PROGRAM FermentationProcess_001
VAR
	

	//MCC Driver	
	fbDriveReverse_001		      : FB_DriveReverse;
	fbDriveReverse_002		      : FB_DriveReverse;
	fbDriveReverse_003		      : FB_DriveReverse;
	fbDriveReverse_004		      : FB_DriveReverse;
	fbDriveReverse_005		      : FB_DriveReverse;
	fbDriveReverse_006		      : FB_DriveReverse;
	fbDriveReverse_007		      : FB_DriveReverse;
	fbDriveReverse_008		      : FB_DriveReverse;
	fbDriveReverse_009		      : FB_DriveReverse;
	fbDriveReverse_010		      : FB_DriveReverse;
	fbDriveReverse_011		      : FB_DriveReverse;
	fbDriveReverse_012		      : FB_DriveReverse;
	fbDriveReverse_013		      : FB_DriveReverse;
	fbDriveReverse_014		      : FB_DriveReverse;
	fbDriveReverse_015		      : FB_DriveReverse;
	fbDriveReverse_016		      : FB_DriveReverse;
	fbDriveReverse_017		      : FB_DriveReverse;
	fbDriveReverse_018		      : FB_DriveReverse;
	fbDriveReverse_019		      : FB_DriveReverse;
	fbDriveReverse_020		      : FB_DriveReverse;


	//MCC Driver Control
	fbMccRev_001			 	  : FB_MotorControlReverse(fbDriveReverse_001);
	fbMccRev_002			 	  : FB_MotorControlReverse(fbDriveReverse_002);
	fbMccRev_003			 	  : FB_MotorControlReverse(fbDriveReverse_003);
	fbMccRev_004 	 			  : FB_MotorControlReverse(fbDriveReverse_004);
	fbMccRev_005			 	  : FB_MotorControlReverse(fbDriveReverse_005);
	fbMccRev_006			 	  : FB_MotorControlReverse(fbDriveReverse_006);
	fbMccRev_007				  : FB_MotorControlReverse(fbDriveReverse_007);
	fbMccRev_008 	 			  : FB_MotorControlReverse(fbDriveReverse_008);
	fbMccRev_009 	  			  : FB_MotorControlReverse(fbDriveReverse_009);
	fbMccRev_010 	              : FB_MotorControlReverse(fbDriveReverse_010);
	fbMccRev_011			 	  : FB_MotorControlReverse(fbDriveReverse_011);
	fbMccRev_012			 	  : FB_MotorControlReverse(fbDriveReverse_012);
	fbMccRev_013			 	  : FB_MotorControlReverse(fbDriveReverse_013);
	fbMccRev_014 	 			  : FB_MotorControlReverse(fbDriveReverse_014);
	fbMccRev_015			 	  : FB_MotorControlReverse(fbDriveReverse_015);
	fbMccRev_016			 	  : FB_MotorControlReverse(fbDriveReverse_016);
	fbMccRev_017				  : FB_MotorControlReverse(fbDriveReverse_017);
	fbMccRev_018 	 			  : FB_MotorControlReverse(fbDriveReverse_018);
	fbMccRev_019 	  			  : FB_MotorControlReverse(fbDriveReverse_019);
	fbMccRev_020 	              : FB_MotorControlReverse(fbDriveReverse_020);
	
	//Temperature Sensor
	fbTempSens_001				  : FB_Scaling;
	fbTempSens_002				  : FB_Scaling;
	fbTempSens_003				  : FB_Scaling;
	//Level Sensor
	fbLevelSens_001				  : FB_Scaling;
	//Ph Sensor
	fbPhSens_001				  : FB_Scaling;	
	//Pressure Sensor
	fbPressureSens_001			  : FB_Scaling;	
	
	
	
	
	
END_VAR

ACT_Motor();
ACT_TempSens();
ACT_LevelSens();
ACT_PhSens();

ACTION ACT_LevelSens:
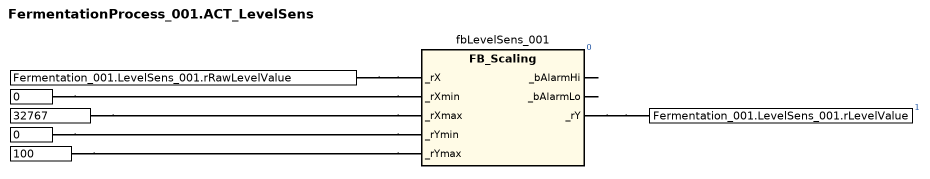
fbLevelSens_001(
    _rX := Fermentation_001.LevelSens_001.rRawLevelValue,
    _rXmin := 0,
    _rXmax := 32767,
    _rYmin := 0,
    _rYmax := 100); // FB_Scaling
Fermentation_001.LevelSens_001.rLevelValue := fbLevelSens_001._rY;
END_ACTION

ACTION ACT_Motor:
//Sygnały obiektów MccRev_* mieszadeł fermentora

//***************************************************SCADA********************************************************

//MccRev_001 variable sets by SCADA
FermentationProcess_001.fbMccRev_001.ScadaAutoButton     := Fermentation_001.MccRev_001.bAutoButton;    // SCADA button Auto Command
FermentationProcess_001.fbMccRev_001.ScadaForwardButton  := Fermentation_001.MccRev_001.bForwardButton; // SCADA button Forward Command
FermentationProcess_001.fbMccRev_001.ScadaReverseButton  := Fermentation_001.MccRev_001.bReverseButton; // SCADA button Reverse Command

//MccRev_002 variable sets by SCADA
FermentationProcess_001.fbMccRev_002.ScadaAutoButton     := Fermentation_001.MccRev_002.bAutoButton;    // SCADA button Auto Command
FermentationProcess_001.fbMccRev_002.ScadaForwardButton  := Fermentation_001.MccRev_002.bForwardButton; // SCADA button Forward Command
FermentationProcess_001.fbMccRev_002.ScadaReverseButton  := Fermentation_001.MccRev_002.bReverseButton; // SCADA button Reverse Command

//MccRev_003 variable sets by SCADA
FermentationProcess_001.fbMccRev_003.ScadaAutoButton     := Fermentation_001.MccRev_003.bAutoButton;    // SCADA button Auto Command
FermentationProcess_001.fbMccRev_003.ScadaForwardButton  := Fermentation_001.MccRev_003.bForwardButton; // SCADA button Forward Command
FermentationProcess_001.fbMccRev_003.ScadaReverseButton  := Fermentation_001.MccRev_003.bReverseButton; // SCADA button Reverse Command

//MccRev_004 variable sets by SCADA
FermentationProcess_001.fbMccRev_004.ScadaAutoButton     := Fermentation_001.MccRev_004.bAutoButton;    // SCADA button Auto Command
FermentationProcess_001.fbMccRev_004.ScadaForwardButton  := Fermentation_001.MccRev_004.bForwardButton; // SCADA button Forward Command
FermentationProcess_001.fbMccRev_004.ScadaReverseButton  := Fermentation_001.MccRev_004.bReverseButton; // SCADA button Reverse Command

//MccRev_005 variable sets by SCADA
FermentationProcess_001.fbMccRev_005.ScadaAutoButton     := Fermentation_001.MccRev_005.bAutoButton;    // SCADA button Auto Command
FermentationProcess_001.fbMccRev_005.ScadaForwardButton  := Fermentation_001.MccRev_005.bForwardButton; // SCADA button Forward Command
FermentationProcess_001.fbMccRev_005.ScadaReverseButton  := Fermentation_001.MccRev_005.bReverseButton; // SCADA button Reverse Command

//MccRev_006 variable sets by SCADA
FermentationProcess_001.fbMccRev_006.ScadaAutoButton     := Fermentation_001.MccRev_006.bAutoButton;    // SCADA button Auto Command
FermentationProcess_001.fbMccRev_006.ScadaForwardButton  := Fermentation_001.MccRev_006.bForwardButton; // SCADA button Forward Command
FermentationProcess_001.fbMccRev_006.ScadaReverseButton  := Fermentation_001.MccRev_006.bReverseButton; // SCADA button Reverse Command

//MccRev_007 variable sets by SCADA
FermentationProcess_001.fbMccRev_007.ScadaAutoButton     := Fermentation_001.MccRev_007.bAutoButton;    // SCADA button Auto Command
FermentationProcess_001.fbMccRev_007.ScadaForwardButton  := Fermentation_001.MccRev_007.bForwardButton; // SCADA button Forward Command
FermentationProcess_001.fbMccRev_007.ScadaReverseButton  := Fermentation_001.MccRev_007.bReverseButton; // SCADA button Reverse Command

//MccRev_008 variable sets by SCADA
FermentationProcess_001.fbMccRev_008.ScadaAutoButton     := Fermentation_001.MccRev_008.bAutoButton;    // SCADA button Auto Command
FermentationProcess_001.fbMccRev_008.ScadaForwardButton  := Fermentation_001.MccRev_008.bForwardButton; // SCADA button Forward Command
FermentationProcess_001.fbMccRev_008.ScadaReverseButton  := Fermentation_001.MccRev_008.bReverseButton; // SCADA button Reverse Command

//MccRev_009 variable sets by SCADA
FermentationProcess_001.fbMccRev_009.ScadaAutoButton     := Fermentation_001.MccRev_009.bAutoButton;    // SCADA button Auto Command
FermentationProcess_001.fbMccRev_009.ScadaForwardButton  := Fermentation_001.MccRev_009.bForwardButton; // SCADA button Forward Command
FermentationProcess_001.fbMccRev_009.ScadaReverseButton  := Fermentation_001.MccRev_009.bReverseButton; // SCADA button Reverse Command

//MccRev_010 variable sets by SCADA
FermentationProcess_001.fbMccRev_010.ScadaAutoButton     := Fermentation_001.MccRev_010.bAutoButton;    // SCADA button Auto Command
FermentationProcess_001.fbMccRev_010.ScadaForwardButton  := Fermentation_001.MccRev_010.bForwardButton; // SCADA button Forward Command
FermentationProcess_001.fbMccRev_010.ScadaReverseButton  := Fermentation_001.MccRev_010.bReverseButton; // SCADA button Reverse Command

//MccRev_011 variable sets by SCADA
FermentationProcess_001.fbMccRev_011.ScadaAutoButton     := Fermentation_001.MccRev_011.bAutoButton;    // SCADA button Auto Command
FermentationProcess_001.fbMccRev_011.ScadaForwardButton  := Fermentation_001.MccRev_011.bForwardButton; // SCADA button Forward Command
FermentationProcess_001.fbMccRev_011.ScadaReverseButton  := Fermentation_001.MccRev_011.bReverseButton; // SCADA button Reverse Command

//MccRev_012 variable sets by SCADA
FermentationProcess_001.fbMccRev_012.ScadaAutoButton     := Fermentation_001.MccRev_012.bAutoButton;    // SCADA button Auto Command
FermentationProcess_001.fbMccRev_012.ScadaForwardButton  := Fermentation_001.MccRev_012.bForwardButton; // SCADA button Forward Command
FermentationProcess_001.fbMccRev_012.ScadaReverseButton  := Fermentation_001.MccRev_012.bReverseButton; // SCADA button Reverse Command

//MccRev_013 variable sets by SCADA
FermentationProcess_001.fbMccRev_013.ScadaAutoButton     := Fermentation_001.MccRev_013.bAutoButton;    // SCADA button Auto Command
FermentationProcess_001.fbMccRev_013.ScadaForwardButton  := Fermentation_001.MccRev_013.bForwardButton; // SCADA button Forward Command
FermentationProcess_001.fbMccRev_013.ScadaReverseButton  := Fermentation_001.MccRev_013.bReverseButton; // SCADA button Reverse Command

//MccRev_014 variable sets by SCADA
FermentationProcess_001.fbMccRev_014.ScadaAutoButton     := Fermentation_001.MccRev_014.bAutoButton;    // SCADA button Auto Command
FermentationProcess_001.fbMccRev_014.ScadaForwardButton  := Fermentation_001.MccRev_014.bForwardButton; // SCADA button Forward Command
FermentationProcess_001.fbMccRev_014.ScadaReverseButton  := Fermentation_001.MccRev_014.bReverseButton; // SCADA button Reverse Command

//MccRev_015 variable sets by SCADA
FermentationProcess_001.fbMccRev_015.ScadaAutoButton     := Fermentation_001.MccRev_015.bAutoButton;    // SCADA button Auto Command
FermentationProcess_001.fbMccRev_015.ScadaForwardButton  := Fermentation_001.MccRev_015.bForwardButton; // SCADA button Forward Command
FermentationProcess_001.fbMccRev_015.ScadaReverseButton  := Fermentation_001.MccRev_015.bReverseButton; // SCADA button Reverse Command

//MccRev_016 variable sets by SCADA
FermentationProcess_001.fbMccRev_016.ScadaAutoButton     := Fermentation_001.MccRev_016.bAutoButton;    // SCADA button Auto Command
FermentationProcess_001.fbMccRev_016.ScadaForwardButton  := Fermentation_001.MccRev_016.bForwardButton; // SCADA button Forward Command
FermentationProcess_001.fbMccRev_016.ScadaReverseButton  := Fermentation_001.MccRev_016.bReverseButton; // SCADA button Reverse Command

//MccRev_017 variable sets by SCADA
FermentationProcess_001.fbMccRev_017.ScadaAutoButton     := Fermentation_001.MccRev_017.bAutoButton;    // SCADA button Auto Command
FermentationProcess_001.fbMccRev_017.ScadaForwardButton  := Fermentation_001.MccRev_017.bForwardButton; // SCADA button Forward Command
FermentationProcess_001.fbMccRev_017.ScadaReverseButton  := Fermentation_001.MccRev_017.bReverseButton; // SCADA button Reverse Command

//MccRev_018 variable sets by SCADA
FermentationProcess_001.fbMccRev_018.ScadaAutoButton     := Fermentation_001.MccRev_018.bAutoButton;    // SCADA button Auto Command
FermentationProcess_001.fbMccRev_018.ScadaForwardButton  := Fermentation_001.MccRev_018.bForwardButton; // SCADA button Forward Command
FermentationProcess_001.fbMccRev_018.ScadaReverseButton  := Fermentation_001.MccRev_018.bReverseButton; // SCADA button Reverse Command

//MccRev_019 variable sets by SCADA
FermentationProcess_001.fbMccRev_019.ScadaAutoButton     := Fermentation_001.MccRev_019.bAutoButton;    // SCADA button Auto Command
FermentationProcess_001.fbMccRev_019.ScadaForwardButton  := Fermentation_001.MccRev_019.bForwardButton; // SCADA button Forward Command
FermentationProcess_001.fbMccRev_019.ScadaReverseButton  := Fermentation_001.MccRev_019.bReverseButton; // SCADA button Reverse Command

//MccRev_020 variable sets by SCADA
FermentationProcess_001.fbMccRev_020.ScadaAutoButton     := Fermentation_001.MccRev_020.bAutoButton;    // SCADA button Auto Command
FermentationProcess_001.fbMccRev_020.ScadaForwardButton  := Fermentation_001.MccRev_020.bForwardButton; // SCADA button Forward Command
FermentationProcess_001.fbMccRev_020.ScadaReverseButton  := Fermentation_001.MccRev_020.bReverseButton; // SCADA button Reverse Command


//***************************************************PLC********************************************************************


//MccRev_001 variable sets by PLC
FermentationProcess_001.fbDriveReverse_001.MotorProtection := Fermentation_001.MccRev_001.bTermFuse;       // PLC input thermal fuse
Fermentation_001.MccRev_001.bContactor     := FermentationProcess_001.fbDriveReverse_001.MotorContactor;   // PLC output contactor
Fermentation_001.MccRev_001.udHours        := FermentationProcess_001.fbDriveReverse_001.Hours;            // PLC Work Time Counter - hours nonvolatile memory register
Fermentation_001.MccRev_001.uMinutes       := FermentationProcess_001.fbDriveReverse_001.Minuts;           // PLC Work Time Counter - minutes nonvolatile memory register
Fermentation_001.MccRev_001.uSeconds       := FermentationProcess_001.fbDriveReverse_001.Seconds;          // PLC Work Time Counter - seconds nonvolatile memory register
Fermentation_001.MccRev_001.sState         := FermentationProcess_001.fbDriveReverse_001.MotorState;       // PLC Work Time Counter - minutes nonvolatile memory register
Fermentation_001.MccRev_001.sStatus        := FermentationProcess_001.fbDriveReverse_001.MotorStatus;      // PLC Work Time Counter - seconds nonvolatile memory register


//MccRev_002 variable sets by PLC
FermentationProcess_001.fbDriveReverse_002.MotorProtection := Fermentation_001.MccRev_002.bTermFuse;       // PLC input thermal fuse
Fermentation_001.MccRev_002.bContactor     := FermentationProcess_001.fbDriveReverse_002.MotorContactor;   // PLC output contactor
Fermentation_001.MccRev_002.udHours        := FermentationProcess_001.fbDriveReverse_002.Hours;            // PLC Work Time Counter - hours nonvolatile memory register
Fermentation_001.MccRev_002.uMinutes       := FermentationProcess_001.fbDriveReverse_002.Minuts;           // PLC Work Time Counter - minutes nonvolatile memory register
Fermentation_001.MccRev_002.uSeconds       := FermentationProcess_001.fbDriveReverse_002.Seconds;          // PLC Work Time Counter - seconds nonvolatile memory register
Fermentation_001.MccRev_002.sState         := FermentationProcess_001.fbDriveReverse_002.MotorState;       // PLC Work Time Counter - minutes nonvolatile memory register
Fermentation_001.MccRev_002.sStatus        := FermentationProcess_001.fbDriveReverse_002.MotorStatus;      // PLC Work Time Counter - seconds nonvolatile memory register

//MccRev_003 variable sets by PLC
FermentationProcess_001.fbDriveReverse_003.MotorProtection :=Fermentation_001.MccRev_003.bTermFuse;       // PLC input thermal fuse
Fermentation_001.MccRev_003.bContactor     := FermentationProcess_001.fbDriveReverse_003.MotorContactor;   // PLC output contactor
Fermentation_001.MccRev_003.udHours        := FermentationProcess_001.fbDriveReverse_003.Hours;            // PLC Work Time Counter - hours nonvolatile memory register
Fermentation_001.MccRev_003.uMinutes       := FermentationProcess_001.fbDriveReverse_003.Minuts;           // PLC Work Time Counter - minutes nonvolatile memory register
Fermentation_001.MccRev_003.uSeconds       := FermentationProcess_001.fbDriveReverse_003.Seconds;          // PLC Work Time Counter - seconds nonvolatile memory register
Fermentation_001.MccRev_003.sState         := FermentationProcess_001.fbDriveReverse_003.MotorState;       // PLC Work Time Counter - minutes nonvolatile memory register
Fermentation_001.MccRev_003.sStatus        := FermentationProcess_001.fbDriveReverse_003.MotorStatus;      // PLC Work Time Counter - seconds nonvolatile memory register

//MccRev_004 variable sets by PLC
FermentationProcess_001.fbDriveReverse_004.MotorProtection := Fermentation_001.MccRev_004.bTermFuse;       // PLC input thermal fuse
Fermentation_001.MccRev_004.bContactor     := FermentationProcess_001.fbDriveReverse_004.MotorContactor;   // PLC output contactor
Fermentation_001.MccRev_004.udHours        := FermentationProcess_001.fbDriveReverse_004.Hours;            // PLC Work Time Counter - hours nonvolatile memory register
Fermentation_001.MccRev_004.uMinutes       := FermentationProcess_001.fbDriveReverse_004.Minuts;           // PLC Work Time Counter - minutes nonvolatile memory register
Fermentation_001.MccRev_004.uSeconds       := FermentationProcess_001.fbDriveReverse_004.Seconds;          // PLC Work Time Counter - seconds nonvolatile memory register
Fermentation_001.MccRev_004.sState         := FermentationProcess_001.fbDriveReverse_004.MotorState;       // PLC Work Time Counter - minutes nonvolatile memory register
Fermentation_001.MccRev_004.sStatus        := FermentationProcess_001.fbDriveReverse_004.MotorStatus;      // PLC Work Time Counter - seconds nonvolatile memory register


//MccRev_005 variable sets by PLC
FermentationProcess_001.fbDriveReverse_005.MotorProtection := Fermentation_001.MccRev_005.bTermFuse;       // PLC input thermal fuse
Fermentation_001.MccRev_005.bContactor     := FermentationProcess_001.fbDriveReverse_005.MotorContactor;   // PLC output contactor
Fermentation_001.MccRev_005.udHours        := FermentationProcess_001.fbDriveReverse_005.Hours;            // PLC Work Time Counter - hours nonvolatile memory register
Fermentation_001.MccRev_005.uMinutes       := FermentationProcess_001.fbDriveReverse_005.Minuts;           // PLC Work Time Counter - minutes nonvolatile memory register
Fermentation_001.MccRev_005.uSeconds       := FermentationProcess_001.fbDriveReverse_005.Seconds;          // PLC Work Time Counter - seconds nonvolatile memory register
Fermentation_001.MccRev_005.sState         := FermentationProcess_001.fbDriveReverse_005.MotorState;       // PLC Work Time Counter - minutes nonvolatile memory register
Fermentation_001.MccRev_005.sStatus        := FermentationProcess_001.fbDriveReverse_005.MotorStatus;      // PLC Work Time Counter - seconds nonvolatile memory register


//MccRev_006 variable sets by PLC
FermentationProcess_001.fbDriveReverse_006.MotorProtection := Fermentation_001.MccRev_006.bTermFuse;       // PLC input thermal fuse
Fermentation_001.MccRev_006.bContactor     := FermentationProcess_001.fbDriveReverse_006.MotorContactor;   // PLC output contactor
Fermentation_001.MccRev_006.udHours        := FermentationProcess_001.fbDriveReverse_006.Hours;            // PLC Work Time Counter - hours nonvolatile memory register
Fermentation_001.MccRev_006.uMinutes       := FermentationProcess_001.fbDriveReverse_006.Minuts;           // PLC Work Time Counter - minutes nonvolatile memory register
Fermentation_001.MccRev_006.uSeconds       := FermentationProcess_001.fbDriveReverse_006.Seconds;          // PLC Work Time Counter - seconds nonvolatile memory register
Fermentation_001.MccRev_006.sState         := FermentationProcess_001.fbDriveReverse_006.MotorState;       // PLC Work Time Counter - minutes nonvolatile memory register
Fermentation_001.MccRev_006.sStatus        := FermentationProcess_001.fbDriveReverse_006.MotorStatus;      // PLC Work Time Counter - seconds nonvolatile memory register

//MccRev_007 variable sets by PLC
FermentationProcess_001.fbDriveReverse_007.MotorProtection := Fermentation_001.MccRev_007.bTermFuse;       // PLC input thermal fuse
Fermentation_001.MccRev_007.bContactor     := FermentationProcess_001.fbDriveReverse_007.MotorContactor;   // PLC output contactor
Fermentation_001.MccRev_007.udHours        := FermentationProcess_001.fbDriveReverse_007.Hours;            // PLC Work Time Counter - hours nonvolatile memory register
Fermentation_001.MccRev_007.uMinutes       := FermentationProcess_001.fbDriveReverse_007.Minuts;           // PLC Work Time Counter - minutes nonvolatile memory register
Fermentation_001.MccRev_007.uSeconds       := FermentationProcess_001.fbDriveReverse_007.Seconds;          // PLC Work Time Counter - seconds nonvolatile memory register
Fermentation_001.MccRev_007.sState         := FermentationProcess_001.fbDriveReverse_007.MotorState;       // PLC Work Time Counter - minutes nonvolatile memory register
Fermentation_001.MccRev_007.sStatus        := FermentationProcess_001.fbDriveReverse_007.MotorStatus;      // PLC Work Time Counter - seconds nonvolatile memory register

//MccRev_008 variable sets by PLC
FermentationProcess_001.fbDriveReverse_008.MotorProtection := Fermentation_001.MccRev_008.bTermFuse;       // PLC input thermal fuse
Fermentation_001.MccRev_008.bContactor     := FermentationProcess_001.fbDriveReverse_008.MotorContactor;   // PLC output contactor
Fermentation_001.MccRev_008.udHours        := FermentationProcess_001.fbDriveReverse_008.Hours;            // PLC Work Time Counter - hours nonvolatile memory register
Fermentation_001.MccRev_008.uMinutes       := FermentationProcess_001.fbDriveReverse_008.Minuts;           // PLC Work Time Counter - minutes nonvolatile memory register
Fermentation_001.MccRev_008.uSeconds       := FermentationProcess_001.fbDriveReverse_008.Seconds;          // PLC Work Time Counter - seconds nonvolatile memory register
Fermentation_001.MccRev_008.sState         := FermentationProcess_001.fbDriveReverse_008.MotorState;       // PLC Work Time Counter - minutes nonvolatile memory register
Fermentation_001.MccRev_008.sStatus        := FermentationProcess_001.fbDriveReverse_008.MotorStatus;      // PLC Work Time Counter - seconds nonvolatile memory register


//MccRev_009 variable sets by PLC
FermentationProcess_001.fbDriveReverse_009.MotorProtection := Fermentation_001.MccRev_009.bTermFuse;       // PLC input thermal fuse
Fermentation_001.MccRev_009.bContactor     := FermentationProcess_001.fbDriveReverse_009.MotorContactor;   // PLC output contactor
Fermentation_001.MccRev_009.udHours        := FermentationProcess_001.fbDriveReverse_009.Hours;            // PLC Work Time Counter - hours nonvolatile memory register
Fermentation_001.MccRev_009.uMinutes       := FermentationProcess_001.fbDriveReverse_009.Minuts;           // PLC Work Time Counter - minutes nonvolatile memory register
Fermentation_001.MccRev_009.uSeconds       := FermentationProcess_001.fbDriveReverse_009.Seconds;          // PLC Work Time Counter - seconds nonvolatile memory register
Fermentation_001.MccRev_009.sState         := FermentationProcess_001.fbDriveReverse_009.MotorState;       // PLC Work Time Counter - minutes nonvolatile memory register
Fermentation_001.MccRev_009.sStatus        := FermentationProcess_001.fbDriveReverse_009.MotorStatus;      // PLC Work Time Counter - seconds nonvolatile memory register

//MccRev_010 variable sets by PLC
FermentationProcess_001.fbDriveReverse_010.MotorProtection := Fermentation_001.MccRev_010.bTermFuse;       // PLC input thermal fuse
Fermentation_001.MccRev_010.bContactor     := FermentationProcess_001.fbDriveReverse_010.MotorContactor;   // PLC output contactor
Fermentation_001.MccRev_010.udHours        := FermentationProcess_001.fbDriveReverse_010.Hours;            // PLC Work Time Counter - hours nonvolatile memory register
Fermentation_001.MccRev_010.uMinutes       := FermentationProcess_001.fbDriveReverse_010.Minuts;           // PLC Work Time Counter - minutes nonvolatile memory register
Fermentation_001.MccRev_010.uSeconds       := FermentationProcess_001.fbDriveReverse_010.Seconds;          // PLC Work Time Counter - seconds nonvolatile memory register
Fermentation_001.MccRev_010.sState         := FermentationProcess_001.fbDriveReverse_010.MotorState;       // PLC Work Time Counter - minutes nonvolatile memory register
Fermentation_001.MccRev_010.sStatus        := FermentationProcess_001.fbDriveReverse_010.MotorStatus;      // PLC Work Time Counter - seconds nonvolatile memory register

//MccRev_011 variable sets by PLC
FermentationProcess_001.fbDriveReverse_011.MotorProtection := Fermentation_001.MccRev_011.bTermFuse;       // PLC input thermal fuse
Fermentation_001.MccRev_011.bContactor     := FermentationProcess_001.fbDriveReverse_011.MotorContactor;   // PLC output contactor
Fermentation_001.MccRev_011.udHours        := FermentationProcess_001.fbDriveReverse_011.Hours;            // PLC Work Time Counter - hours nonvolatile memory register
Fermentation_001.MccRev_011.uMinutes       := FermentationProcess_001.fbDriveReverse_011.Minuts;           // PLC Work Time Counter - minutes nonvolatile memory register
Fermentation_001.MccRev_011.uSeconds       := FermentationProcess_001.fbDriveReverse_011.Seconds;          // PLC Work Time Counter - seconds nonvolatile memory register
Fermentation_001.MccRev_011.sState         := FermentationProcess_001.fbDriveReverse_011.MotorState;       // PLC Work Time Counter - minutes nonvolatile memory register
Fermentation_001.MccRev_011.sStatus        := FermentationProcess_001.fbDriveReverse_011.MotorStatus;      // PLC Work Time Counter - seconds nonvolatile memory register


//MccRev_012 variable sets by PLC
FermentationProcess_001.fbDriveReverse_012.MotorProtection := Fermentation_001.MccRev_012.bTermFuse;       // PLC input thermal fuse
Fermentation_001.MccRev_012.bContactor     := FermentationProcess_001.fbDriveReverse_012.MotorContactor;   // PLC output contactor
Fermentation_001.MccRev_012.udHours        := FermentationProcess_001.fbDriveReverse_012.Hours;            // PLC Work Time Counter - hours nonvolatile memory register
Fermentation_001.MccRev_012.uMinutes       := FermentationProcess_001.fbDriveReverse_012.Minuts;           // PLC Work Time Counter - minutes nonvolatile memory register
Fermentation_001.MccRev_012.uSeconds       := FermentationProcess_001.fbDriveReverse_012.Seconds;          // PLC Work Time Counter - seconds nonvolatile memory register
Fermentation_001.MccRev_012.sState         := FermentationProcess_001.fbDriveReverse_012.MotorState;       // PLC Work Time Counter - minutes nonvolatile memory register
Fermentation_001.MccRev_012.sStatus        := FermentationProcess_001.fbDriveReverse_012.MotorStatus;      // PLC Work Time Counter - seconds nonvolatile memory register


//MccRev_013 variable sets by PLC
FermentationProcess_001.fbDriveReverse_013.MotorProtection := Fermentation_001.MccRev_013.bTermFuse;       // PLC input thermal fuse
Fermentation_001.MccRev_013.bContactor     := FermentationProcess_001.fbDriveReverse_013.MotorContactor;   // PLC output contactor
Fermentation_001.MccRev_013.udHours        := FermentationProcess_001.fbDriveReverse_013.Hours;            // PLC Work Time Counter - hours nonvolatile memory register
Fermentation_001.MccRev_013.uMinutes       := FermentationProcess_001.fbDriveReverse_013.Minuts;           // PLC Work Time Counter - minutes nonvolatile memory register
Fermentation_001.MccRev_013.uSeconds       := FermentationProcess_001.fbDriveReverse_013.Seconds;          // PLC Work Time Counter - seconds nonvolatile memory register
Fermentation_001.MccRev_013.sState         := FermentationProcess_001.fbDriveReverse_013.MotorState;       // PLC Work Time Counter - minutes nonvolatile memory register
Fermentation_001.MccRev_013.sStatus        := FermentationProcess_001.fbDriveReverse_013.MotorStatus;      // PLC Work Time Counter - seconds nonvolatile memory register


//MccRev_014 variable sets by PLC
FermentationProcess_001.fbDriveReverse_014.MotorProtection := Fermentation_001.MccRev_014.bTermFuse;       // PLC input thermal fuse
Fermentation_001.MccRev_014.bContactor     := FermentationProcess_001.fbDriveReverse_014.MotorContactor;   // PLC output contactor
Fermentation_001.MccRev_014.udHours        := FermentationProcess_001.fbDriveReverse_014.Hours;            // PLC Work Time Counter - hours nonvolatile memory register
Fermentation_001.MccRev_014.uMinutes       := FermentationProcess_001.fbDriveReverse_014.Minuts;           // PLC Work Time Counter - minutes nonvolatile memory register
Fermentation_001.MccRev_014.uSeconds       := FermentationProcess_001.fbDriveReverse_014.Seconds;          // PLC Work Time Counter - seconds nonvolatile memory register
Fermentation_001.MccRev_014.sState         := FermentationProcess_001.fbDriveReverse_014.MotorState;       // PLC Work Time Counter - minutes nonvolatile memory register
Fermentation_001.MccRev_014.sStatus        := FermentationProcess_001.fbDriveReverse_014.MotorStatus;      // PLC Work Time Counter - seconds nonvolatile memory register

//MccRev_015 variable sets by PLC
FermentationProcess_001.fbDriveReverse_015.MotorProtection := Fermentation_001.MccRev_015.bTermFuse;       // PLC input thermal fuse
Fermentation_001.MccRev_015.bContactor     := FermentationProcess_001.fbDriveReverse_015.MotorContactor;   // PLC output contactor
Fermentation_001.MccRev_015.udHours        := FermentationProcess_001.fbDriveReverse_015.Hours;            // PLC Work Time Counter - hours nonvolatile memory register
Fermentation_001.MccRev_015.uMinutes       := FermentationProcess_001.fbDriveReverse_015.Minuts;           // PLC Work Time Counter - minutes nonvolatile memory register
Fermentation_001.MccRev_015.uSeconds       := FermentationProcess_001.fbDriveReverse_015.Seconds;          // PLC Work Time Counter - seconds nonvolatile memory register
Fermentation_001.MccRev_015.sState         := FermentationProcess_001.fbDriveReverse_015.MotorState;       // PLC Work Time Counter - minutes nonvolatile memory register
Fermentation_001.MccRev_015.sStatus        := FermentationProcess_001.fbDriveReverse_015.MotorStatus;      // PLC Work Time Counter - seconds nonvolatile memory register


//MccRev_016 variable sets by PLC
FermentationProcess_001.fbDriveReverse_016.MotorProtection := Fermentation_001.MccRev_016.bTermFuse;       // PLC input thermal fuse
Fermentation_001.MccRev_016.bContactor     := FermentationProcess_001.fbDriveReverse_016.MotorContactor;   // PLC output contactor
Fermentation_001.MccRev_016.udHours        := FermentationProcess_001.fbDriveReverse_016.Hours;            // PLC Work Time Counter - hours nonvolatile memory register
Fermentation_001.MccRev_016.uMinutes       := FermentationProcess_001.fbDriveReverse_016.Minuts;           // PLC Work Time Counter - minutes nonvolatile memory register
Fermentation_001.MccRev_016.uSeconds       := FermentationProcess_001.fbDriveReverse_016.Seconds;          // PLC Work Time Counter - seconds nonvolatile memory register
Fermentation_001.MccRev_016.sState         := FermentationProcess_001.fbDriveReverse_016.MotorState;       // PLC Work Time Counter - minutes nonvolatile memory register
Fermentation_001.MccRev_016.sStatus        := FermentationProcess_001.fbDriveReverse_016.MotorStatus;      // PLC Work Time Counter - seconds nonvolatile memory register


//MccRev_017 variable sets by PLC
FermentationProcess_001.fbDriveReverse_017.MotorProtection := Fermentation_001.MccRev_017.bTermFuse;       // PLC input thermal fuse
Fermentation_001.MccRev_017.bContactor     := FermentationProcess_001.fbDriveReverse_017.MotorContactor;   // PLC output contactor
Fermentation_001.MccRev_017.udHours        := FermentationProcess_001.fbDriveReverse_017.Hours;            // PLC Work Time Counter - hours nonvolatile memory register
Fermentation_001.MccRev_017.uMinutes       := FermentationProcess_001.fbDriveReverse_017.Minuts;           // PLC Work Time Counter - minutes nonvolatile memory register
Fermentation_001.MccRev_017.uSeconds       := FermentationProcess_001.fbDriveReverse_017.Seconds;          // PLC Work Time Counter - seconds nonvolatile memory register
Fermentation_001.MccRev_017.sState         := FermentationProcess_001.fbDriveReverse_017.MotorState;       // PLC Work Time Counter - minutes nonvolatile memory register
Fermentation_001.MccRev_017.sStatus        := FermentationProcess_001.fbDriveReverse_017.MotorStatus;      // PLC Work Time Counter - seconds nonvolatile memory register


//MccRev_018 variable sets by PLC
FermentationProcess_001.fbDriveReverse_018.MotorProtection := Fermentation_001.MccRev_018.bTermFuse;       // PLC input thermal fuse
Fermentation_001.MccRev_018.bContactor     := FermentationProcess_001.fbDriveReverse_018.MotorContactor;   // PLC output contactor
Fermentation_001.MccRev_018.udHours        := FermentationProcess_001.fbDriveReverse_018.Hours;            // PLC Work Time Counter - hours nonvolatile memory register
Fermentation_001.MccRev_018.uMinutes       := FermentationProcess_001.fbDriveReverse_018.Minuts;           // PLC Work Time Counter - minutes nonvolatile memory register
Fermentation_001.MccRev_018.uSeconds       := FermentationProcess_001.fbDriveReverse_018.Seconds;          // PLC Work Time Counter - seconds nonvolatile memory register
Fermentation_001.MccRev_018.sState         := FermentationProcess_001.fbDriveReverse_018.MotorState;       // PLC Work Time Counter - minutes nonvolatile memory register
Fermentation_001.MccRev_018.sStatus        := FermentationProcess_001.fbDriveReverse_018.MotorStatus;      // PLC Work Time Counter - seconds nonvolatile memory register


//MccRev_019 variable sets by PLC
FermentationProcess_001.fbDriveReverse_019.MotorProtection := Fermentation_001.MccRev_019.bTermFuse;       // PLC input thermal fuse
Fermentation_001.MccRev_019.bContactor     := FermentationProcess_001.fbDriveReverse_019.MotorContactor;   // PLC output contactor
Fermentation_001.MccRev_019.udHours        := FermentationProcess_001.fbDriveReverse_019.Hours;            // PLC Work Time Counter - hours nonvolatile memory register
Fermentation_001.MccRev_019.uMinutes       := FermentationProcess_001.fbDriveReverse_019.Minuts;           // PLC Work Time Counter - minutes nonvolatile memory register
Fermentation_001.MccRev_019.uSeconds       := FermentationProcess_001.fbDriveReverse_019.Seconds;          // PLC Work Time Counter - seconds nonvolatile memory register
Fermentation_001.MccRev_019.sState         := FermentationProcess_001.fbDriveReverse_019.MotorState;       // PLC Work Time Counter - minutes nonvolatile memory register
Fermentation_001.MccRev_019.sStatus        := FermentationProcess_001.fbDriveReverse_019.MotorStatus;      // PLC Work Time Counter - seconds nonvolatile memory register


//MccRev_020 variable sets by PLC
FermentationProcess_001.fbDriveReverse_020.MotorProtection := Fermentation_001.MccRev_020.bTermFuse;       // PLC input thermal fuse
Fermentation_001.MccRev_020.bContactor     := FermentationProcess_001.fbDriveReverse_020.MotorContactor;   // PLC output contactor
Fermentation_001.MccRev_020.udHours        := FermentationProcess_001.fbDriveReverse_020.Hours;            // PLC Work Time Counter - hours nonvolatile memory register
Fermentation_001.MccRev_020.uMinutes       := FermentationProcess_001.fbDriveReverse_020.Minuts;           // PLC Work Time Counter - minutes nonvolatile memory register
Fermentation_001.MccRev_020.uSeconds       := FermentationProcess_001.fbDriveReverse_020.Seconds;          // PLC Work Time Counter - seconds nonvolatile memory register
Fermentation_001.MccRev_020.sState         := FermentationProcess_001.fbDriveReverse_020.MotorState;       // PLC Work Time Counter - minutes nonvolatile memory register
Fermentation_001.MccRev_020.sStatus        := FermentationProcess_001.fbDriveReverse_020.MotorStatus;      // PLC Work Time Counter - seconds nonvolatile memory register
END_ACTION

ACTION ACT_PhSens:
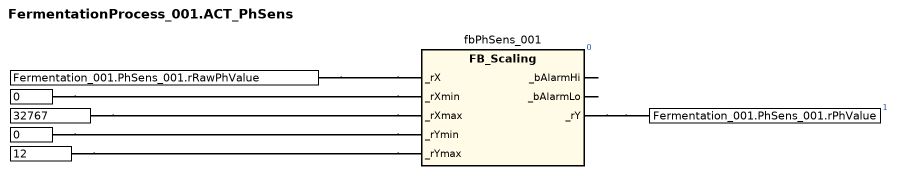
fbPhSens_001(
    _rX := Fermentation_001.PhSens_001.rRawPhValue,
    _rXmin := 0,
    _rXmax := 32767,
    _rYmin := 0,
    _rYmax := 12); // FB_Scaling
Fermentation_001.PhSens_001.rPhValue := fbPhSens_001._rY;
END_ACTION

ACTION ACT_PressureSens:
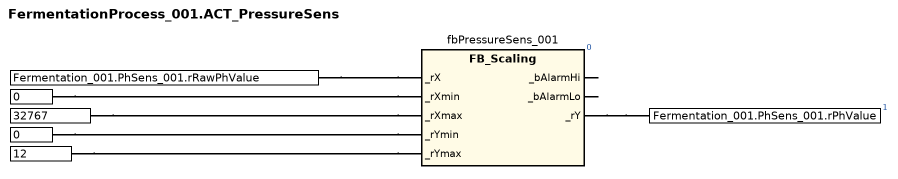
fbPressureSens_001(
    _rX := Fermentation_001.PhSens_001.rRawPhValue,
    _rXmin := 0,
    _rXmax := 32767,
    _rYmin := 0,
    _rYmax := 12); // FB_Scaling
Fermentation_001.PhSens_001.rPhValue := fbPressureSens_001._rY;
END_ACTION

ACTION ACT_TempSens:
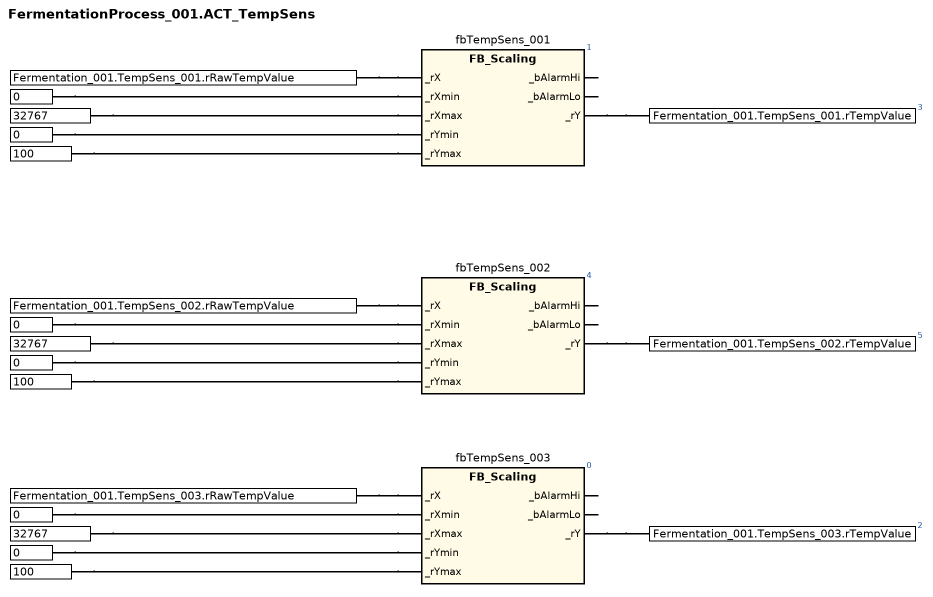
fbTempSens_003(
    _rX := Fermentation_001.TempSens_003.rRawTempValue,
    _rXmin := 0,
    _rXmax := 32767,
    _rYmin := 0,
    _rYmax := 100); // FB_Scaling
fbTempSens_001(
    _rX := Fermentation_001.TempSens_001.rRawTempValue,
    _rXmin := 0,
    _rXmax := 32767,
    _rYmin := 0,
    _rYmax := 100); // FB_Scaling
Fermentation_001.TempSens_003.rTempValue := fbTempSens_003._rY;
Fermentation_001.TempSens_001.rTempValue := fbTempSens_001._rY;
fbTempSens_002(
    _rX := Fermentation_001.TempSens_002.rRawTempValue,
    _rXmin := 0,
    _rXmax := 32767,
    _rYmin := 0,
    _rYmax := 100); // FB_Scaling
Fermentation_001.TempSens_002.rTempValue := fbTempSens_002._rY;
END_ACTION

END_PROGRAM

(* stored: Version 1.1.0.1, ProductVersion 3.1.4024.12
   POU FermentationProcess_001: Id {cd4debd5-e4da-4fbd-a7f2-abb66eea5825}, SpecialFunc None
   Action ACT_LevelSens: Id {8ee61bea-2bee-417e-8d54-d51a566be6b4}
   Action ACT_Motor: Id {7e5ca941-1b2f-4bd8-a7e6-7c6d33833563}
   Action ACT_PhSens: Id {c132ae7c-f82a-406c-b89d-8bb7114273eb}
   Action ACT_PressureSens: Id {6ccb0a22-bf81-4ede-881e-cab4baf9ffd0}
   Action ACT_TempSens: Id {1c3023f9-db11-40ae-aa02-b0cabd6dbc52} *)
